{attribute 'GeneratedUsingTerminal: EK1110-0043-0016'}
{attribute addProperty BoxType "EK1110-0043-0016"}
{attribute addProperty Id "EtcSlaveTerminalBaseInfoDataAT %I*InfoData_6F19DB2B2"}
{attribute addProperty CRC "2874840167"}
{attribute addProperty Size "2"}
TYPE EK1110_AB5A9467 EXTENDS EtcSlaveTerminalBase :
STRUCT
	{attribute addProperty Name "InfoData"}
	InfoData : InfoData_6F19DB2B;
END_STRUCT
END_TYPE

(* stored: Version 1.2.0.0, ProductVersion 3.1.4024.9
   DUT EK1110_AB5A9467: Id {40ed625b-22ec-4df4-857f-6f46ebd219bb} *)
